RoboDK station: ALTERNATIVA 1 - PYTHON.rdk

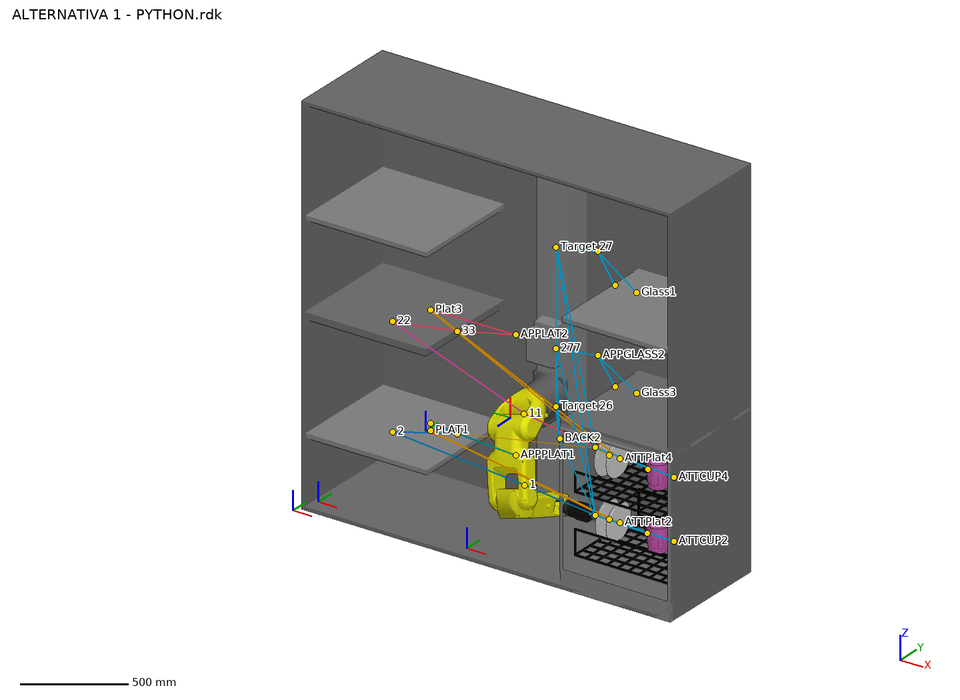
[picture v0: the station drawn from its stored meshes, robots at their saved joint values, targets as dots, program paths as lines]
Station ALTERNATIVA 1 (saved by RoboDK 6.0.0). Poses are relative to the parent item; angles as X-Y-Z fixed-axis rotations.
  - object dishwasher_system_concept_v8_widebay_without_doors at (0, 0, 0) mm, size 2080 x 656 x 2100 mm, geometry from dishwasher_system_concept_v8_widebay_without_doors.obj
  - frame MUEBLE  at (-14.91, -46.19, 5.82) mm
  - frame Frame 3 at (0, 1000, 0) mm
  - frame Frame 3 at (80, 23.81, 50) mm
    - frame My Mechanism Base at (890, -76.19, 40) mm
      - robot My Mechanism: 1 axes
          modified DH rows (alpha deg, a mm, theta deg, d mm): 0, 0, 0, 0 linear
          base shift (0, 0, 0) mm, rotated rx 180 ry 0 rz 180 deg
          joint limits [0] to [2000]; home [0]; saved at [512.4]
        - frame Fanuc LR Mate 200iD Base at (-120, 180, 120) mm, rotated rx -90 ry 0 rz -180 deg
          - robot Fanuc LR Mate 200iD: 6 axes, payload 7 kg, reach 717 mm, repeatability 0.02 mm, weight 25 kg
              modified DH rows (alpha deg, a mm, theta deg, d mm): 0, 0, 0, 330; -90, 50, -90, 0; 0, 330, 0, 0; -90, 35, 0, 335; 90, 0, 0, 0; -90, 0, 0, 80
              base shift (0, 0, -330) mm
              joint limits [-170, -100, -67, -190, -125, -360] to [170, 145, 213, 190, 124, 360]; home [0, 0, 0, 0, 0, 0]; saved at [-164.543, 69.279, -71.12, 75.946, 84.831, -203.46]
            - tool RobotiQ EPick Vacuum Gripper (1 Cup), TCP at (0, 0, 130) mm, size 75 x 83 x 136.1 mm
    - target ATTCUP4 (Cartesian target) at (1799.24, 294.21, 511.76) mm, rotated rx 89.5 ry -5.17 rz 90.44 deg; joints [-117.93, 89.2, -41.04, -140.24, -48.1, -34.02, 657.02] of Fanuc LR Mate 200iD
    - target ATTCUP2 (Cartesian target) at (1799.24, 294.21, 181.19) mm, rotated rx 89.5 ry -5.17 rz 90.44 deg; joints [-117.93, 89.2, -41.04, -140.24, -48.1, -34.02, 326.45] of Fanuc LR Mate 200iD
    - target ATTCUP3 (Cartesian target) at (1652.24, 294.21, 511.76) mm, rotated rx 89.5 ry -5.17 rz 90.44 deg; joints [-138.704, 89.045, -41.226, -119.334, -60.265, -46.149, 842.02] of Fanuc LR Mate 200iD
    - target ATT CUP1 (Cartesian target) at (1649.27, 294.13, 181.19) mm, rotated rx 89.49 ry -5.15 rz 90.44 deg; joints [-139.659, 91.138, -38.735, -117.247, -59.734, -49.065, 524.79] of Fanuc LR Mate 200iD
    - target ATTPlat4 (Cartesian target) at (1492.24, 294.21, 521.76) mm, rotated rx 89.5 ry -5.17 rz 90.44 deg; joints [-150.545, 73.908, -62.326, -115.936, -76.644, -29.865, 842.02] of Fanuc LR Mate 200iD
    - target ATTPlat3 (Cartesian target) at (1435.24, 294.21, 521.76) mm, rotated rx 89.5 ry -5.17 rz 90.44 deg; joints [-155.939, 71.504, -66.631, -111.67, -80.507, -26.808, 842.02] of Fanuc LR Mate 200iD
    - target ATTPlat2 (Cartesian target) at (1492.29, 294.17, 192.18) mm, rotated rx 89.49 ry -5.16 rz 90.45 deg; joints [-150.54, 73.9, -62.32, -115.93, -76.64, -29.86, 512.4] of Fanuc LR Mate 200iD
    - target ATTPlat1 (Cartesian target) at (1433.29, 294.17, 192.18) mm, rotated rx 89.49 ry -5.16 rz 90.45 deg; joints [-156.132, 71.426, -66.759, -111.499, -80.626, -26.706, 512.4] of Fanuc LR Mate 200iD
    - target APPLevel1 (Cartesian target) at (1353.29, 294.17, 192.18) mm, rotated rx 89.49 ry -5.16 rz 90.45 deg; joints [-164.543, 69.279, -71.12, -104.054, -84.831, -23.46, 512.4] of Fanuc LR Mate 200iD
    - target AppLevel2 (Cartesian target) at (1353.31, 294.13, 539.32) mm, rotated rx 89.49 ry -5.16 rz 90.45 deg; joints [-164.54, 69.27, -71.12, -104.05, -84.83, -23.46, 859.5] of Fanuc LR Mate 200iD
    - target PLAT1 (Cartesian target) at (428.51, 290.58, 368.19) mm, rotated rx 179.22 ry -5.15 rz 90.44 deg; joints [118.577, 88.107, -38.029, -103.762, -65.066, -49.818, 735.54] of Fanuc LR Mate 200iD
    - target APPPLAT1 (Cartesian target) at (907.77, 293.69, 374.71) mm, rotated rx 179.22 ry -5.15 rz 90.44 deg; joints [161.39, 59.852, -97.065, -160.717, -91.517, 2.711, 735.54] of Fanuc LR Mate 200iD
    - target 1 (Cartesian target) at (1105.92, 79.49, 363.07) mm, rotated rx 177.16 ry -5.16 rz 90.45 deg; joints [-164.212, 13.105, -61.63, -15.411, 57.28, -172.522, 714.88] of Fanuc LR Mate 200iD
    - target 2 (joint target) at (954.3, -768.06, 933.65) mm, rotated rx -87.4 ry 4.4 rz 178.42 deg; joints [36.79, -3.451, 75.152, -0.663, 11.706, 123.069, 698.35] of Fanuc LR Mate 200iD
    - target 3 (Cartesian target) at (1048.68, -378.27, 793.15) mm, rotated rx -37.81 ry -5.8 rz -90.22 deg; joints [161.38, 59.85, 93.11, -160.71, -91.51, 2.71, 735.54] of Fanuc LR Mate 200iD
    - target Plat2 (Cartesian target) at (428.51, 290.58, 370.19) mm, rotated rx 179.22 ry -5.15 rz 90.44 deg; joints [118.426, 87.858, -38.318, -103.786, -65.25, -49.54, 735.54] of Fanuc LR Mate 200iD
    - target 11 (Cartesian target) at (1104.33, 79.48, 729.5) mm, rotated rx 177.14 ry -5.16 rz 90.46 deg; joints [-163.5, 10.533, -62.557, -16.069, 58.261, -172.441, 1061.98] of Fanuc LR Mate 200iD
    - target 22 (joint target) at (954.29, -768.07, 1499.8) mm, rotated rx -87.39 ry 4.38 rz 178.42 deg; joints [36.78, -3.441, 75.162, -0.665, 11.686, 123.081, 1264.46] of Fanuc LR Mate 200iD
    - target 33 (Cartesian target) at (1048.68, -378.27, 1322.07) mm, rotated rx -37.81 ry -5.8 rz -90.22 deg; joints [161.38, 59.85, 93.11, -160.71, -91.51, 2.71, 1264.46] of Fanuc LR Mate 200iD
    - target Plat3 (Cartesian target) at (428.41, 290.49, 988.07) mm, rotated rx 179.23 ry -5.15 rz 90.46 deg; joints [118.57, 88.1, -38.02, -103.76, -65.06, -49.81, 1355.37] of Fanuc LR Mate 200iD
    - target APPLAT2 (Cartesian target) at (907.77, 293.68, 994.57) mm, rotated rx 179.22 ry -5.15 rz 90.44 deg; joints [161.39, 59.85, -97.07, -160.72, -91.52, 2.71, 1355.37] of Fanuc LR Mate 200iD
    - target Plat4 (Cartesian target) at (428.41, 290.49, 990.07) mm, rotated rx 179.23 ry -5.15 rz 90.46 deg; joints [118.418, 87.851, -38.308, -103.783, -65.245, -49.532, 1355.37] of Fanuc LR Mate 200iD
    - target APPPLATLEVL1 (Cartesian target) at (428.51, 290.58, 408.19) mm, rotated rx 179.22 ry -5.15 rz 90.44 deg; joints [115.465, 83.932, -42.984, -103.564, -68.538, -45.19, 735.54] of Fanuc LR Mate 200iD
    - target APPPLATLEVEL2 (Cartesian target) at (428.41, 290.49, 990.07) mm, rotated rx 179.23 ry -5.15 rz 90.46 deg; joints [118.418, 87.851, -38.308, -103.783, -65.245, -49.532, 1355.37] of Fanuc LR Mate 200iD
    - target BACK2 (Cartesian target) at (1154.28, 293.48, 529.25) mm, rotated rx 177.09 ry -5.16 rz 90.45 deg; joints [-154.571, 59.952, -100.067, -22.513, 94.125, -183.666, 859.5] of Fanuc LR Mate 200iD
    - target Target 26 (Cartesian target) at (1145.8, 278.18, 697.85) mm, rotated rx 177.09 ry -5.16 rz 90.45 deg; joints [-131.988, 67.786, -129.675, -49.71, 112.279, -209.086, 859.5] of Fanuc LR Mate 200iD
    - target Target 27 (Cartesian target) at (1145.88, 278.21, 1518.83) mm, rotated rx 177.08 ry -5.17 rz 90.45 deg; joints [-131.97, 67.78, -129.67, -49.71, 112.26, -209.08, 1680.44] of Fanuc LR Mate 200iD
    - target Glass1 (Cartesian target) at (1594.18, 283.21, 1408.63) mm, rotated rx 91.31 ry -5.16 rz 90.45 deg; joints [-131.692, 67.533, -70.233, 42.242, 74.516, -198.295, 1586.78] of Fanuc LR Mate 200iD
    - target AppGlass (Cartesian target) at (1388.67, 267.22, 1567.61) mm, rotated rx 91.31 ry -5.16 rz 90.45 deg; joints [-135.941, 60.631, -112.337, 46.701, 105.143, -169.095, 1586.78] of Fanuc LR Mate 200iD
    - target Glass2 (Cartesian target) at (1476.25, 282.04, 1411.33) mm, rotated rx 91.31 ry -5.16 rz 90.45 deg; joints [-142.218, 62.552, -83.009, 51.173, 85.031, -190.594, 1586.78] of Fanuc LR Mate 200iD
    - target 277 (Cartesian target) at (1145.84, 278.18, 995.38) mm, rotated rx 177.09 ry -5.16 rz 90.45 deg; joints [-131.98, 67.78, -129.67, -49.71, 112.27, -209.08, 1157.02] of Fanuc LR Mate 200iD
    - target APPGLASS2 (Cartesian target) at (1388.7, 267.22, 1033.15) mm, rotated rx 91.31 ry -5.15 rz 90.45 deg; joints [-135.94, 60.63, -112.33, 46.7, 105.14, -169.09, 1052.34] of Fanuc LR Mate 200iD
    - target Glass3 (Cartesian target) at (1594.2, 283.2, 890.72) mm, rotated rx 91.32 ry -5.16 rz 90.46 deg; joints [-131.69, 67.53, -70.23, 42.24, 74.51, -198.29, 1068.87] of Fanuc LR Mate 200iD
    - target Glass4 (Cartesian target) at (1476.23, 282.03, 893.4) mm, rotated rx 91.32 ry -5.16 rz 90.45 deg; joints [-142.22, 62.55, -83.01, 51.17, 85.03, -190.59, 1068.87] of Fanuc LR Mate 200iD
  - program MainProgram (2 instructions, listed below)
  - program RecallPosition (3 instructions, listed below)
  - program Attach (3 instructions, listed below)
  - program SwitchSide (8 instructions, listed below)
  - program SwitchSide2 (8 instructions, listed below)
  - program BacktoSide (8 instructions, listed below)
  - program BackToSide2 (8 instructions, listed below)
  - program Plates (29 instructions, listed below)
  - program Detach (3 instructions, listed below)
  - program Glass (48 instructions, listed below)
  - object PLATO2 at (1520, 300, 260) mm, rotated rx -90 ry 0 rz 90 deg, size 200 x 200 x 4 mm, geometry from tinker.obj
  - object PLATO3 at (1580, 300, 260) mm, rotated rx -90 ry 0 rz 90 deg, size 200 x 200 x 4 mm, geometry from tinker.obj
  - object PLATO at (1521.8, 288.65, 590) mm, rotated rx -90 ry 0 rz 90 deg, size 200 x 200 x 4 mm, geometry from tinker.obj
  - object PLATO1 at (1580, 300, 590) mm, rotated rx -90 ry 0 rz 90 deg, size 200 x 200 x 4 mm, geometry from tinker.obj
  - object VASO_1 at (1800, 320, 485) mm, rotated rx 90 ry 0 rz 0 deg, size 110.6 x 132.4 x 110.6 mm, geometry from glass-obj.obj
  - object VASO_2 at (1950, 320, 485) mm, rotated rx 90 ry 0 rz 0 deg, size 110.6 x 132.4 x 110.6 mm, geometry from glass-obj.obj
  - object VASO_3 at (1800, 320, 159) mm, rotated rx 90 ry 0 rz 0 deg, size 110.6 x 132.4 x 110.6 mm, geometry from glass-obj.obj
  - object VASO_4 at (1950, 320, 159) mm, rotated rx 90 ry 0 rz 0 deg, size 110.6 x 132.4 x 110.6 mm, geometry from glass-obj.obj
  - Python program Prog11 (listed below)
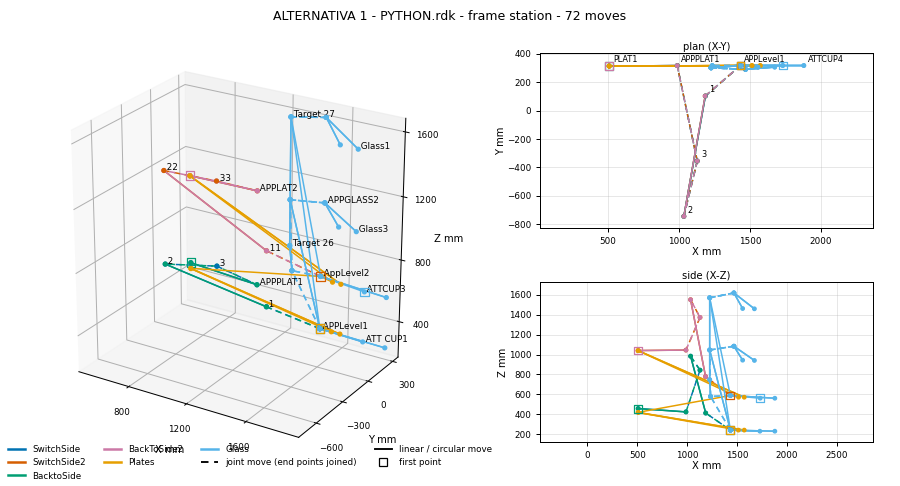
[picture p0: tool path of ALTERNATIVA 1 - PYTHON.rdk in frame station, 72 of 72 moves have a stored position in this frame; points joined in program order, loops and branches not executed]

--- program MainProgram (robot Fanuc LR Mate 200iD) ---
  Call Plates
  Call Glass

--- program RecallPosition (robot Fanuc LR Mate 200iD) ---
  Set Ref.: Frame 3
  Set Tool: RobotiQ EPick Vacuum Gripper (1 Cup)
  Move objects

--- program Attach (robot Fanuc LR Mate 200iD) ---
  Set Ref.: Frame 3
  Set Tool: RobotiQ EPick Vacuum Gripper (1 Cup)
  Attach to RobotiQ EPick Vacuum Gripper (1 Cup)

--- program SwitchSide (robot Fanuc LR Mate 200iD) ---
  Set Ref.: Frame 3
  Set Tool: RobotiQ EPick Vacuum Gripper (1 Cup)
  MoveL (APPLevel1)
  MoveJ (1)
  MoveL (2)
  MoveJ (3)
  MoveJ (APPPLAT1)
  MoveL (APPPLATLEVL1)

--- program SwitchSide2 (robot Fanuc LR Mate 200iD) ---
  Set Ref.: Frame 3
  Set Tool: RobotiQ EPick Vacuum Gripper (1 Cup)
  MoveL (AppLevel2)
  MoveJ (11)
  MoveL (22)
  MoveJ (33)
  MoveJ (APPLAT2)
  MoveL (APPPLATLEVEL2)

--- program BacktoSide (robot Fanuc LR Mate 200iD) ---
  Set Ref.: Frame 3
  Set Tool: RobotiQ EPick Vacuum Gripper (1 Cup)
  MoveL (APPPLATLEVL1)
  MoveL (APPPLAT1)
  MoveJ (3)
  MoveJ (2)
  MoveL (1)
  MoveJ (APPLevel1)

--- program BackToSide2 (robot Fanuc LR Mate 200iD) ---
  Set Ref.: Frame 3
  Set Tool: RobotiQ EPick Vacuum Gripper (1 Cup)
  MoveL (APPPLATLEVEL2)
  MoveL (APPLAT2)
  MoveJ (33)
  MoveJ (22)
  MoveL (11)
  MoveJ (AppLevel2)

--- program Plates (robot Fanuc LR Mate 200iD) ---
  Set Ref.: Frame 3
  Set Tool: RobotiQ EPick Vacuum Gripper (1 Cup)
  MoveJ (APPLevel1)
  MoveL (ATTPlat1)
  Call Attach
  Call SwitchSide
  MoveL (PLAT1)
  Call Detach
  Call BacktoSide
  MoveL (ATTPlat2)
  Call Attach
  Call Attach
  Call SwitchSide
  MoveL (Plat2)
  Call Detach
  Call BacktoSide
  MoveL (AppLevel2)
  MoveL (ATTPlat3)
  Call Attach
  Call SwitchSide2
  MoveL (Plat3)
  Call Detach
  Call BackToSide2
  MoveL (ATTPlat4)
  Call Attach
  Call SwitchSide2
  MoveL (Plat4)
  Call Detach
  Call BackToSide2

--- program Detach (robot Fanuc LR Mate 200iD) ---
  Set Ref.: Frame 3
  Set Tool: RobotiQ EPick Vacuum Gripper (1 Cup)
  Detach from RobotiQ EPick Vacuum Gripper (1 Cup)

--- program Glass (robot Fanuc LR Mate 200iD) ---
  Set Ref.: Frame 3
  Set Tool: RobotiQ EPick Vacuum Gripper (1 Cup)
  MoveL (ATTCUP3)
  Call Attach
  MoveL (AppLevel2)
  MoveJ (BACK2)
  MoveL (Target 26)
  MoveL (Target 27)
  MoveJ (AppGlass)
  MoveL (Glass1)
  Call Detach
  MoveL (AppGlass)
  MoveJ (Target 27)
  MoveL (AppLevel2)
  MoveL (ATTCUP4)
  Call Attach
  MoveL (AppLevel2)
  MoveJ (BACK2)
  MoveL (Target 26)
  MoveL (Target 27)
  MoveJ (AppGlass)
  MoveL (Glass2)
  Call Detach
  MoveL (AppGlass)
  MoveJ (Target 27)
  MoveL (APPLevel1)
  MoveL (ATT CUP1)
  Call Attach
  MoveL (APPLevel1)
  MoveJ (BACK2)
  MoveJ (277)
  MoveJ (APPGLASS2)
  MoveL (Glass3)
  Call Detach
  MoveL (APPGLASS2)
  MoveJ (277)
  MoveL (APPLevel1)
  MoveL (ATTCUP2)
  Call Attach
  MoveL (APPLevel1)
  MoveJ (BACK2)
  MoveJ (277)
  MoveJ (APPGLASS2)
  MoveL (Glass4)
  Call Detach
  MoveL (APPGLASS2)
  MoveJ (277)
  MoveL (APPLevel1)

--- Python program Prog11 ---
# ============================================================
# ANALISIS ROBODK - MainProgram = Plates + Glass
#
# Datos mostrados:
# - Programa analizado
# - Tiempo ciclo
# - Distancia recorrida por el TCP en mm y m
# - Instrucciones válidas
# - Total de instrucciones
# - Total de movimientos
# - Nº MoveJ
# - Nº MoveL
# ============================================================

import os
import csv
import datetime

try:
    from robodk.robolink import *
except:
    from robolink import *


# ================= CONFIGURACIÓN =================

PROGRAMA_PRINCIPAL = "MainProgram"

SUBPROGRAMAS = [
    "Plates",
    "Glass"
]

EXPORTAR_CSV = True


# ================= CONEXIÓN CON ROBODK =================

RDK = Robolink()


def obtener_programa(nombre):
    prog = RDK.Item(nombre, ITEM_TYPE_PROGRAM)

    if not prog.Valid():
        RDK.ShowMessage("No se ha encontrado el programa: " + nombre)
        raise Exception("No se ha encontrado el programa: " + nombre)

    return prog


programa_principal = obtener_programa(PROGRAMA_PRINCIPAL)

programas_sub = []

for nombre in SUBPROGRAMAS:
    programas_sub.append(obtener_programa(nombre))


# ================= TIEMPO, DISTANCIA E INSTRUCCIONES VÁLIDAS =================
#
# Como MainProgram llama a Plates y Glass, el movimiento real está dentro
# de Plates y Glass.
#
# Por eso:
# Tiempo ciclo = tiempo Plates + tiempo Glass
# Distancia TCP = distancia Plates + distancia Glass
# Instrucciones válidas = válidas Plates + válidas Glass

tiempo_ciclo_total_s = 0.0
distancia_tcp_total_mm = 0.0
instrucciones_validas_total = 0

for prog in programas_sub:

    try:
        resultado_update = prog.Update(COLLISION_ON, 3600)

        instrucciones_validas = int(resultado_update[0])
        tiempo_ciclo_s = float(resultado_update[1])
        distancia_tcp_mm = float(resultado_update[2])

    except Exception as e:
        instrucciones_validas = 0
        tiempo_ciclo_s = 0.0
        distancia_tcp_mm = 0.0
        RDK.ShowMessage("Error al actualizar el programa " + prog.Name() + ": " + str(e))

    instrucciones_validas_total += instrucciones_validas
    tiempo_ciclo_total_s += tiempo_ciclo_s
    distancia_tcp_total_mm += distancia_tcp_mm


distancia_tcp_total_m = distancia_tcp_total_mm / 1000.0


# ================= CONTAR INSTRUCCIONES Y MOVIMIENTOS =================
#
# Aquí contamos:
# MainProgram + Plates + Glass
#
# MainProgram tendrá normalmente las llamadas a Plates y Glass.
# Plates y Glass tendrán los movimientos reales.

programas_a_contar = [programa_principal] + programas_sub

total_instrucciones = 0
total_movimientos = 0
num_movej = 0
num_movel = 0

for prog in programas_a_contar:

    n_instr = prog.InstructionCount()
    total_instrucciones += n_instr

    for i in range(n_instr):

        try:
            nombre, instype, movetype, es_target_articular, pose, joints = prog.Instruction(i)
        except:
            continue

        if instype == INS_TYPE_MOVE:

            total_movimientos += 1

            if movetype == MOVE_TYPE_JOINT:
                num_movej += 1

            elif movetype == MOVE_TYPE_LINEAR:
                num_movel += 1


# ================= MOSTRAR RESULTADOS =================

nombre_analisis = PROGRAMA_PRINCIPAL + " = " + " + ".join(SUBPROGRAMAS)

mensaje = ""
mensaje += "RESULTADOS DEL PROGRAMA ROBODK\n"
mensaje += "====================================\n\n"

mensaje += "Programa analizado: {}\n".format(nombre_analisis)
mensaje += "Tiempo ciclo: {:.3f} s\n".format(tiempo_ciclo_total_s)
mensaje += "Distancia recorrida por el TCP: {:.3f} mm\n".format(distancia_tcp_total_mm)
mensaje += "Distancia recorrida por el TCP: {:.3f} m\n".format(distancia_tcp_total_m)
mensaje += "Instrucciones válidas: {}\n".format(instrucciones_validas_total)
mensaje += "Total de instrucciones: {}\n".format(total_instrucciones)
mensaje += "Total de movimientos: {}\n".format(total_movimientos)
mensaje += "Nº MoveJ: {}\n".format(num_movej)
mensaje += "Nº MoveL: {}\n".format(num_movel)

print(mensaje)
RDK.ShowMessage(mensaje)


# ================= EXPORTAR A CSV =================

if EXPORTAR_CSV:

    escritorio = os.path.join(os.path.expanduser("~"), "Desktop")
    ruta_csv = os.path.join(escritorio, "resultados_robodk_MainProgram.csv")

    if not os.path.isdir(escritorio):
        ruta_csv = os.path.join(os.getcwd(), "resultados_robodk_MainProgram.csv")

    existe_archivo = os.path.isfile(ruta_csv)

    with open(ruta_csv, mode="a", newline="", encoding="utf-8-sig") as archivo:
        writer = csv.writer(archivo, delimiter=";")

        if not existe_archivo:
            writer.writerow([
                "Fecha",
                "Programa analizado",
                "Tiempo ciclo (s)",
                "Distancia TCP (mm)",
                "Distancia TCP (m)",
                "Instrucciones validas",
                "Total instrucciones",
                "Total movimientos",
                "MoveJ",
                "MoveL"
            ])

        writer.writerow([
            datetime.datetime.now().strftime("%Y-%m-%d %H:%M:%S"),
            nombre_analisis,
            round(tiempo_ciclo_total_s, 3),
            round(distancia_tcp_total_mm, 3),
            round(distancia_tcp_total_m, 3),
            instrucciones_validas_total,
            total_instrucciones,
            total_movimientos,
            num_movej,
            num_movel
        ])

    print("\nCSV guardado en:")
    print(ruta_csv)
